(* CoDeSys 2.3 export: ATTR4_TU.EXP *)

(* Data type in Diag/Parameter *)
TYPE attr4_tu :
STRUCT
	DefaultValue_as16		: INT;
(*
	DefaultValue_as16		: ARRAY [1..16] OF INT;
	AnalogChannel_as16	: ARRAY [1..16] OF INT;
	Frequency_as16			: ARRAY [1..16] OF INT;
	data_au8 				: ARRAY [1..2] OF USINT;
*)
END_STRUCT
END_TYPE
